TYPE T_HMI_PACK_Barcode : STRING(cMAX_HMI_PACKCODE_LENGHT);
END_TYPE

(* stored: Version 1.1.0.1
   DUT T_HMI_PACK_Barcode: Id {3365de05-84a1-43ca-9f3b-4a66c9670583} *)
